{attribute 'TcGenerated'}
{attribute 'no-analysis'}
{attribute 'linkalways'}
// This function has been automatically generated from the project information.
VAR_GLOBAL CONSTANT
	{attribute 'const_non_replaced'}
	stLibVersion_ApplicationBase : ST_LibVersion := (iMajor := 1, iMinor := 1, iBuild := 0, iRevision := 0, nFlags := 0, sVersion := '1.1.0');
END_VAR

(* stored: Version 1.1.0.1, ProductVersion 3.1.4026.20
   GVL Global_Version: Id {ffd1fff3-c0ef-4501-985f-811a119b50ee} *)
